FUNCTION_BLOCK StatusToStringLogVisitor IMPLEMENTS ITF_Visitor
VAR
	StringLog : reference to T_MaxString;
END_VAR

METHOD FB_init : BOOL
VAR_INPUT
	bInitRetains : BOOL; // if TRUE, the retain variables are initialized (warm start / cold start)
	bInCopyCode : BOOL;  // if TRUE, the instance afterwards gets moved into the copy code (online change)
	StringLog : T_MaxString;
END_VAR
END_METHOD

METHOD VisitBaseObject : BOOL
VAR_INPUT
	BaseObject : ITF_Base;
END_VAR
StringLog := CONCAT(StringLog, '[');
StringLog := CONCAT(StringLog, BaseObject.Name);
StringLog := CONCAT(StringLog, ']');

IF BaseObject.HasError THEN
	StringLog := CONCAT(StringLog, ': Has Error ');
	StringLog := CONCAT(StringLog, BaseObject.GetErrorMessage());
	StringLog := CONCAT(StringLog, '. ');
ELSE
	StringLog := CONCAT(StringLog, ': Has No Error. ');
END_IF
END_METHOD

END_FUNCTION_BLOCK

(* stored: Version 1.1.0.1, ProductVersion 3.1.4024.12
   POU StatusToStringLogVisitor: Id {eba75a34-823b-4e39-abb3-56acdb274577}, SpecialFunc None
   Method FB_init: Id {100c23b1-17ac-4e57-ba7c-e0a63aab2bbe}
   Method VisitBaseObject: Id {153bcbe8-de52-4e13-9ec4-da3b21a98915} *)
